DATA_BLOCK "Plc"
{ S7_Optimized_Access := 'FALSE' }
VERSION : 0.1
NON_RETAIN
   STRUCT
      "1层上行呼梯按钮指示灯" : Bool;
      "2层上行呼梯按钮指示灯" : Bool;
      "3层上行呼梯按钮指示灯" : Bool;
      "4层上行呼梯按钮指示灯" : Bool;
      "5层上行呼梯按钮指示灯" : Bool;
      "6层上行呼梯按钮指示灯" : Bool;
      "7层上行呼梯按钮指示灯" : Bool;
      "8层上行呼梯按钮指示灯" : Bool;
      "9层上行呼梯按钮指示灯" : Bool;
      "2层下行呼梯按钮指示灯" : Bool;
      "3层下行呼梯按钮指示灯" : Bool;
      "4层下行呼梯按钮指示灯" : Bool;
      "5层下行呼梯按钮指示灯" : Bool;
      "6层下行呼梯按钮指示灯" : Bool;
      "7层下行呼梯按钮指示灯" : Bool;
      "8层下行呼梯按钮指示灯" : Bool;
      "9层下行呼梯按钮指示灯" : Bool;
      "10层下行呼梯按钮指示灯" : Bool;
      "1号梯1层按钮指示灯" : Bool;
      "1号梯2层按钮指示灯" : Bool;
      "1号梯3层按钮指示灯" : Bool;
      "1号梯4层按钮指示灯" : Bool;
      "1号梯5层按钮指示灯" : Bool;
      "1号梯6层按钮指示灯" : Bool;
      "1号梯7层按钮指示灯" : Bool;
      "1号梯8层按钮指示灯" : Bool;
      "1号梯9层按钮指示灯" : Bool;
      "1号梯10层按钮指示灯" : Bool;
      "1号梯LEDa" : Bool;
      "1号梯LEDb" : Bool;
      "1号梯LEDc" : Bool;
      "1号梯LEDd" : Bool;
      "1号梯LEDe" : Bool;
      "1号梯LEDf" : Bool;
      "1号梯LEDg" : Bool;
      "1号梯LEDh" : Bool;
      "1号梯LEDi" : Bool;
      "1号梯LEDj" : Bool;
      "1号梯LEDk" : Bool;
      "1号梯LEDl" : Bool;
      "1号梯LEDm" : Bool;
      "1号梯LEDn" : Bool;
      "1号梯上行指示" : Bool;
      "1号梯下行指示" : Bool;
      "1号梯故障指示" : Bool;
      "1号梯照明指示" : Bool;
      "1号梯风扇指示" : Bool;
      "1号梯满载指示" : Bool;
      "1号梯电机启动信号" : Bool;
      "1号梯上行接触器" : Bool;
      "1号梯下行接触器" : Bool;
      "1号梯高速接触器" : Bool;
      "1号梯低速接触器" : Bool;
      "1号梯开门继电器" : Bool;
      "1号梯关门继电器" : Bool;
      "1号梯1级减速制动" : Bool;
      "1号梯2级减速制动" : Bool;
      "1号梯3级减速制动" : Bool;
      "2号梯1层按钮指示灯" : Bool;
      "2号梯2层按钮指示灯" : Bool;
      "2号梯3层按钮指示灯" : Bool;
      "2号梯4层按钮指示灯" : Bool;
      "2号梯5层按钮指示灯" : Bool;
      "2号梯6层按钮指示灯" : Bool;
      "2号梯7层按钮指示灯" : Bool;
      "2号梯8层按钮指示灯" : Bool;
      "2号梯9层按钮指示灯" : Bool;
      "2号梯10层按钮指示灯" : Bool;
      "2号梯LEDa" : Bool;
      "2号梯LEDb" : Bool;
      "2号梯LEDc" : Bool;
      "2号梯LEDd" : Bool;
      "2号梯LEDe" : Bool;
      "2号梯LEDf" : Bool;
      "2号梯LEDg" : Bool;
      "2号梯LEDh" : Bool;
      "2号梯LEDi" : Bool;
      "2号梯LEDj" : Bool;
      "2号梯LEDk" : Bool;
      "2号梯LEDl" : Bool;
      "2号梯LEDm" : Bool;
      "2号梯LEDn" : Bool;
      "2号梯上行指示" : Bool;
      "2号梯下行指示" : Bool;
      "2号梯故障指示" : Bool;
      "2号梯照明指示" : Bool;
      "2号梯风扇指示" : Bool;
      "2号梯满载指示" : Bool;
      "2号梯电机启动信号" : Bool;
      "2号梯上行接触器" : Bool;
      "2号梯下行接触器" : Bool;
      "2号梯高速接触器" : Bool;
      "2号梯低速接触器" : Bool;
      "2号梯开门继电器" : Bool;
      "2号梯关门继电器" : Bool;
      "2号梯1级减速制动" : Bool;
      "2号梯2级减速制动" : Bool;
      "2号梯3级减速制动" : Bool;
      "3号梯1层按钮指示灯" : Bool;
      "3号梯2层按钮指示灯" : Bool;
      "3号梯3层按钮指示灯" : Bool;
      "3号梯4层按钮指示灯" : Bool;
      "3号梯5层按钮指示灯" : Bool;
      "3号梯6层按钮指示灯" : Bool;
      "3号梯7层按钮指示灯" : Bool;
      "3号梯8层按钮指示灯" : Bool;
      "3号梯9层按钮指示灯" : Bool;
      "3号梯10层按钮指示灯" : Bool;
      "3号梯LEDa" : Bool;
      "3号梯LEDb" : Bool;
      "3号梯LEDc" : Bool;
      "3号梯LEDd" : Bool;
      "3号梯LEDe" : Bool;
      "3号梯LEDf" : Bool;
      "3号梯LEDg" : Bool;
      "3号梯LEDh" : Bool;
      "3号梯LEDi" : Bool;
      "3号梯LEDj" : Bool;
      "3号梯LEDk" : Bool;
      "3号梯LEDl" : Bool;
      "3号梯LEDm" : Bool;
      "3号梯LEDn" : Bool;
      "3号梯上行指示" : Bool;
      "3号梯下行指示" : Bool;
      "3号梯故障指示" : Bool;
      "3号梯照明指示" : Bool;
      "3号梯风扇指示" : Bool;
      "3号梯满载指示" : Bool;
      "3号梯电机启动信号" : Bool;
      "3号梯上行接触器" : Bool;
      "3号梯下行接触器" : Bool;
      "3号梯高速接触器" : Bool;
      "3号梯低速接触器" : Bool;
      "3号梯开门继电器" : Bool;
      "3号梯关门继电器" : Bool;
      "3号梯1级减速制动" : Bool;
      "3号梯2级减速制动" : Bool;
      "3号梯3级减速制动" : Bool;
      准备就绪信号 : Bool;
   END_STRUCT;


BEGIN

END_DATA_BLOCK

